// TIA Portal V19 export
TYPE "LEXCHANGETRAY_typeConstraintRollerEm_xPositionAxis_configuration"
// stored: Access Published
   STRUCT
      homeTo1stCellDistance : LReal := 100.0;
      "1stCellTo2ndCellDistance" : LReal := 20.0;
      homeTo1stCellVel : LReal := 20.0;
      "1stCellTo2ndCellVel" : LReal := 10.0;
   END_STRUCT;
END_TYPE
